(* CoDeSys 2.3.9.41 project: CoolingSystem_Simulation.pro *)
(* Libraries: Standard.lib 4.10.05 11:14:46, IecSfc.lib 13.4.06 15:51:28, SYSLIBCALLBACK.LIB 26.9.08 16:43:52 *)

(* Global variable list: Global_Variables *)
VAR_GLOBAL
(*=== INPUTS ===*)
    Start_Button    		  : BOOL;   (* start\stop button *)
    Temp_Inlet      		  : INT;   (* Inlet temperature *)
    Temp_Outlet    		  : INT;   (* Outlet temperature *)
    Pressure_Sensor 	  : INT;  (* Pressure sensor*)
    Water_Level    		  : REAL;  (* Water level sensor *)
    Pump1_FB       		  : BOOL;   (* Pump feedback 1*)
    Pump2_FB        		  : BOOL;  (* Pump feedback 2 *)

(*=== OUTPUTS ===*)
    Pump1_Main          : BOOL;  (* Pump 1 (main) *)
    Pump2_Backup     : BOOL;   (* Pump 2 (backup) *)
    Cooling_Valve         : REAL;   (* Cooling valve *)
    Alarm_Signal   	      : BOOL;   (* Alarm ‘Accident’ *)
    Normal_Op      	      : BOOL;  (* ‘System normal’ signal*)

(*=== SYSTEM STATUS ===*)
    System_Normal       : BOOL;   (* Status ‘System normal’ *)
    System_Alarm        : BOOL;   (* Status ‘Accident’*)
    State_Text     : STRING[50];    (* Current system status *)
    Alarm_Msg : STRING[50]; (* Current alarm message *)
    Button_Txt : STRING[50]; (* Button Start status *)
END_VAR

(* Data type *)
TYPE SystemStates :
STRUCT
END_STRUCT
END_TYPE

(* POU PLC_PRG, ST *)
	PROGRAM PLC_PRG
	(*Main control program for automated temperature and pump management system.
    Handles alarm analysis, pump control, temperature regulation, and system state tracking.*)
	VAR
	    Accident         : BOOL := FALSE;		(* General accident flag *)
	    Temp_Setpoint    : REAL := 120.0;	(* Temperature setpoint (adjustable) *)
	    P_Max            : REAL := 20.0;	 (* Max allowed pressure *)
	    L_Min            : REAL := 10.0;	 (* Min allowed water level *)
	    fbAlarm          : AlarmHandling;	(* Alarm handling block *)
	    fbPump           : PumpControl;	(* Pump control block *)
	    Alarm_Message    : STRING[50];	(* Alarm text message (for HMI) *)
	     fbTempReg : TemperatureRegulation;	(* Temperature regulation block *)
	    Current_State : INT := 0;	(* System state (0-wait, 1-work, 2-alarm) *)
           Mode_Text     : STRING[20];	(* System state as text *)
	    Button_Context  : STRING[50];	 (* Button label (Start/Stop) *)
	END_VAR
	(* --- ALARM handling (checks all key process parameters) --- *)
	fbAlarm(
	    Pressure := Pressure_Sensor,
	    Temp     := Temp_Inlet,
	    Level    := Water_Level,
	    P_Max    := P_Max,
	    T_Max    := Temp_Setpoint,
	    L_Min    := L_Min
	);

	(* --- PUMP control (controls both main and backup, gets status) --- *)
	fbPump(
	    Start      := Start_Button AND NOT fbAlarm.Alarm,	(* Allow start only if no alarm *)
	    FB_Main    := Pump1_FB,
	    FB_Backup  := Pump2_FB
	);

	Pump1_Main   := fbPump.MainPump;
	Pump2_Backup := fbPump.BackupPump;

	(* --- Alarm message logic (priority: pump alarm > process alarm) --- *)
	IF fbPump.Fault THEN
	    Accident := TRUE;
	    Alarm_Signal := TRUE;
	    Alarm_Message := 'Alarm, any pump doesnt working';
	ELSE
		Alarm_Message := fbAlarm.AlarmText;
	END_IF
		Alarm_Msg := Alarm_Message;	(* For HMI (single text variable) *)

	(* --- Temperature regulation block (if system is running and no alarm) --- *)
	IF Start_Button AND NOT fbAlarm.Alarm THEN
	    fbTempReg(
	        Temp_In := Temp_Inlet,
	        Setpoint   := Temp_Setpoint,
	        Kp         := 0.5,
	        Valve_Min  := 0.0,
	        Valve_Max  := 100.0
	    );
	    Cooling_Valve := fbTempReg.Valve_Output;
	ELSE
	    Cooling_Valve := 0.0;	(* Safe default if stopped or alarm *)
	END_IF

	(* --- Global alarm output signal (for lamp/siren) --- *)
	IF fbAlarm.Alarm OR fbPump.Fault THEN
	    Alarm_Signal := TRUE;
	ELSE
	    Alarm_Signal := FALSE;
	END_IF

	(* --- System state machine (0: waiting, 1: working, 2: alarm) --- *)
	IF Alarm_Signal  = TRUE THEN
	    Current_State := 2;
	ELSIF Pump1_Main OR Pump2_Backup THEN
	    Current_State := 1;
	ELSE
	    Current_State := 0;
	END_IF

	(* --- State text for HMI and user feedback --- *)
	CASE Current_State OF
	    0: Mode_Text := 'Waiting';
	    1: Mode_Text := 'Working';
	    2: Mode_Text := 'Accident';
	ELSE
	    Mode_Text := 'Undefined';
	END_CASE

	State_Text := Mode_Text;

	(* --- System flags for HMI LEDs (Normal/Alarm) --- *)
	System_Normal := (Current_State = 1);
	System_Alarm  := (Current_State = 2);

	(* --- Start/Stop button text for HMI context awareness --- *)
	IF Start_Button = FALSE THEN
	Button_Context := 'Start';
	ELSE
	Button_Context := 'Stop';
	END_IF

	Button_Txt := Button_Context;
END_PROGRAM

(* POU AlarmHandling, ST *)
	FUNCTION_BLOCK AlarmHandling
	(*Purpose: Monitors key process parameters (pressure, temperature, water level).
	    If any parameter is out of safe limits, sets Alarm output and descriptive AlarmText.
	    AlarmCode identifies the reason for alarm:
	      1 - High Pressure
	      2 - High Temperature
	      3 - Low Water Level*)
	VAR_INPUT
		Pressure	:	REAL;	 (* Current process pressure *)
		Temp	:	REAL;	(* Current process temperature *)
		Level	:	REAL;	 (* Current water level *)
		P_Max	:	REAL;	(* Maximum allowed pressure *)
		T_Max	:	REAL;	(* Maximum allowed temperature *)
		L_Min	:	REAL;	(* Minimum allowed water level *)
	END_VAR
	VAR_OUTPUT
		Alarm	:	BOOL;	(* Alarm flag, TRUE if any fault detected *)
		AlarmText	:	STRING[50];	(* Description for HMI/operator *)
	END_VAR
	VAR
		AlarmCode	:	INT;	(* Numeric code for alarm reason *)
	END_VAR
	(* Reset alarm status by default *)
	Alarm	:= FALSE;
	AlarmText	:=	' ';
	
	(* Check process limits and set alarm outputs *)
	IF Pressure > P_Max THEN
		Alarm	:=	TRUE;
		AlarmText	:=	'Pressure is higher then normal!';
		AlarmCode	:=	1;
	ELSIF Temp > T_Max	THEN
		Alarm	:=	TRUE;
		AlarmText	:=	'Temterature is higher then normal!';
		AlarmCode	:=	2;
	ELSIF Level < L_Min THEN
		Alarm := TRUE;
		AlarmText	:=	'Alarm, low water level!';
		AlarmCode	:=	3;
	END_IF
END_FUNCTION_BLOCK

(* POU PumpControl, ST *)
	FUNCTION_BLOCK PumpControl
    (*Purpose: Controls main and backup pumps based on start command and feedback signals.
    If main pump feedback is missing, switches to backup pump.
    If both pumps fail, sets Fault output.
    IsBackupOn shows whether backup pump is running.*)
	VAR_INPUT
	    Start        : BOOL;	(* Command to start pumping system *)
	    FB_Main      : BOOL;	(* Feedback from main pump *)
	    FB_Backup    : BOOL;	(* Feedback from backup pump *)
	END_VAR
	
	VAR_OUTPUT
	    MainPump     : BOOL;	(* Output to control main pump *)
	    BackupPump   : BOOL;	(* Output to control backup pump *)
	    Fault        : BOOL;	(* TRUE if neither pump provides feedback *)
	    IsBackupOn   : BOOL;	(* TRUE if backup pump is running *)
	END_VAR

	VAR
	    tryBackup    : BOOL;		(* Internal flag to track switching to backup *)
	END_VAR
	(* Default state: all pumps off, no fault *)
	MainPump   := FALSE;
		BackupPump := FALSE;
		Fault      := FALSE;
		IsBackupOn := FALSE;

	(* Pump control logic *)
	IF Start THEN
	    MainPump := TRUE;
	(* Check main pump feedback *)
	    IF NOT FB_Main THEN
	        BackupPump := TRUE;
	        IsBackupOn := TRUE;

	(* If backup also fails, raise fault *)
	        IF NOT FB_Backup THEN
	            Fault := TRUE;
	        END_IF
	    END_IF
	END_IF
END_FUNCTION_BLOCK

(* POU TemperatureRegulation, ST *)
	FUNCTION_BLOCK TemperatureRegulation
	(* Purpose: Implements a simple proportional temperature control algorithm.
    Adjusts valve position based on error between current temperature and setpoint.
    Output is limited between Valve_Min and Valve_Max.*)
	VAR_INPUT
	    Temp_In   : REAL;	(* Current temperature (sensor value) *)
	    Setpoint     : REAL;	(* Desired target temperature *)
	    Kp           : REAL := 1.0;	(* Proportional gain *)
	    Valve_Min    : REAL := 0.0;	(* Minimum allowed valve position *)
	    Valve_Max    : REAL := 100.0;	(* Maximum allowed valve position *)
	END_VAR

	VAR_OUTPUT
	    Valve_Output : REAL;	(* Output value for the control valve *)
	END_VAR
	
	VAR
	    Error        : REAL;	(* Difference between setpoint and current temperature *)
	    Control      : REAL;	(* Calculated control value *)
	END_VAR
	(* Calculate regulation error *)
	Error := Setpoint - Temp_In;

	(* Proportional control algorithm *)
	Control := Valve_Output + Kp * Error;

	(* Limit output to allowed range (anti-windup) *)
	IF Control > Valve_Max THEN
	    Control := Valve_Max;
	ELSIF Control < Valve_Min THEN
	    Control := Valve_Min;
	END_IF

		Valve_Output := Control;
END_FUNCTION_BLOCK

(* Visualisation MainView
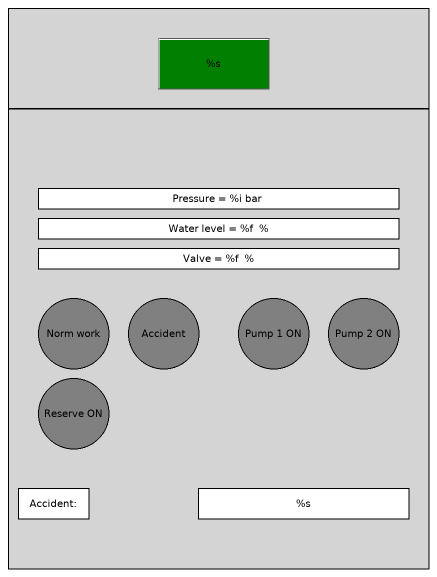
button at (190,60)-(301,111): text "%s"; shows Button_Txt; toggles Start_Button
rectangle at (70,210)-(431,231): text "Pressure = %i bar"; shows Pressure_Sensor; editable 0..1000
rectangle at (70,240)-(431,261): text "Water level = %f  %"; shows Water_Level; editable 0..1000
rectangle at (70,270)-(431,291): text "Valve = %f  %"; shows Cooling_Valve; editable 0..1000
ellipse at (70,320)-(141,391): text "Norm work"; alarm colour if System_Normal
ellipse at (160,320)-(231,391): text "Accident"; alarm colour if System_Alarm
ellipse at (270,320)-(341,391): text "Pump 1 ON"; alarm colour if Pump1_Main
ellipse at (360,320)-(431,391): text "Pump 2 ON"; alarm colour if Pump2_Backup
ellipse at (70,400)-(141,471): text "Reserve ON"; alarm colour if Pump2_Backup
rectangle at (50,510)-(121,541): text "Accident:"
rectangle at (230,510)-(441,541): text "%s"; shows Alarm_Msg
2 more shapes without text or variables
3 elements of other kinds (tables, trends, ...) not read
*)
